PROGRAM Messung1
VAR
	//PWM Settings
	pwmPeriodinSec			: TIME 	:= T#25S;
	pwmDutyCycle			: REAL 	:= 0.0;	
	pwmOutputValveControl 	: FB_PWM;
	status 					: INT 	:= 0; 			//Status 0 : Initial 
													//Status 1 : Heating to Startpoint
													//Status 2 : Heating while recording
													//Status 3 : Cooling while recording
													//STatus is set manuelly
													
END_VAR


(*Temperature should be increased to a value in a first step. 
This is to serve as a 0 point. In the second step, the duty cycle is increased and the step response is recorded.  
The container is then closed. The same duty cycle is used.
Finally, the water is cooled with a DutyCycle of ... .
*)

(* jacket temperature input *)
jacketTempC := INT_TO_REAL(jacketTempRaw)/32768.0*200.0 -50.0;
(* room temperature input *) //Is not in use in TemperaturControl
roomTemp := (INT_TO_REAL(roomTempRaw)/32767.0)*100.0 - 40.0;  (* Sensor Range: -40°C to + 60°C *)



// DutyCycle - To get a startingTemp.
CASE status OF
	
	//------Initial - Status 0----------//
	0:
	(* Setting Valves & Pump off  *)
	pumpOn := FALSE;
	coldValve := FALSE;
	hotValve := FALSE;
	steriValve := FALSE;
	
	//------HEATING - Status 1----------//
	1:
	//Starting pump
	pumpOn := TRUE;
	
	//DutyCyle for startpoint
	pwmDutyCycle:= 20 ;
	pwmOutputValveControl(pwmCycleTime:=pwmPeriodinSec, pwmDutyCycle:=pwmDutyCycle); //Gets the Output
	hotValve := pwmOutputValveControl.Q;
	
	
	//------HEATING - Status 2----------//
	2:	
	//DutyCycle for step response
	pwmDutyCycle:= 40 ;
	pwmOutputValveControl(pwmCycleTime:=pwmPeriodinSec, pwmDutyCycle:=pwmDutyCycle); //Gets the Output
	hotValve := pwmOutputValveControl.Q;
	
	//------COOLING - Status 3----------//
	3:
	//Turning off hotValve
	hotValve := FALSE;
	
	//DutyCycle for cooling
	pwmDutyCycle:= 40 ;
	pwmOutputValveControl(pwmCycleTime:=pwmPeriodinSec, pwmDutyCycle:=pwmDutyCycle); //Gets the Output
	coldValve := pwmOutputValveControl.Q;
END_CASE

END_PROGRAM

(* stored: Version 1.1.0.1, ProductVersion 3.1.4022.12
   POU Messung1: Id {23361215-bda4-4897-81af-964a5b46021b}, SpecialFunc None *)
